Universal Robots URScript: 31-pallet_working.script

def P31pallet_working():
  set_standard_analog_input_domain(0, 1)
  set_standard_analog_input_domain(1, 1)
  set_tool_analog_input_domain(0, 1)
  set_tool_analog_input_domain(1, 1)
  set_analog_outputdomain(0, 0)
  set_analog_outputdomain(1, 0)
  set_tool_voltage(0)
  set_tcp(p[0.0,0.0,0.0,0.0,0.0,0.0])
  set_payload(0.0)
  set_gravity([0.0, 0.0, 9.82])
  global cnt_1=0
  $ 1 "BeforeStart"
  $ 2 "MoveJ"
  $ 3 "home"
  movej([-1.5531271160755855, -1.3695928511239472, -1.6775720824016744, -1.6897506072074169, 1.5962951182804097, 0.016572788116811236], a=1.3962634015954636, v=1.0471975511965976)
  $ 4 "cnt_1≔5"
  global cnt_1=5
  while (True):
    $ 5 "机器人程序"
    $ 6 "托盘"
    cnt_1_x = cnt_1 % 6
    cnt_1_y = floor(cnt_1 / 6)
    u20301u23039_1 = interpolate_pose(interpolate_pose(p[-.099999969066, -.400000054028, .199999960922, -.001221099554, 3.116276478707, .038892320958], p[-.100000003377, -.199999964388, .199999987920, -.001220853457, 3.116276502675, .038892110509], cnt_1_x/5), interpolate_pose(p[.100000089847, -.399999929680, .199999839637, -.001221229174, 3.116276825726, .038892683103], p[.100000030650, -.199999976799, .200000020249, -.001220905867, 3.116276536037, .038892034429],cnt_1_x/5), cnt_1_y/3)
    if (cnt_1 >= 23):
      cnt_1 = 0
    else:
      cnt_1 = cnt_1 + 1
    end
    $ 13 "方式"
    movel(pose_trans(u20301u23039_1, pose_trans(pose_inv(p[-.099999969066, -.400000054028, .199999960922, -.001221099554, 3.116276478707, .038892320958]),p[-.099999970101, -.399999995469, .304818609093, -.001221099554, 3.116276478707, .038892320958])), a=1.2, v=0.25)
    $ 14 "模式点_1"
    movel(u20301u23039_1, a=1.2, v=0.25)
    $ 15 "设置"
    $ 16 "等待: 0"
    $ 17 "退出"
    movel(pose_trans(u20301u23039_1, pose_trans(pose_inv(p[-.099999969066, -.400000054028, .199999960922, -.001221099554, 3.116276478707, .038892320958]),p[-.099999970101, -.399999995469, .304818609093, -.001221099554, 3.116276478707, .038892320958])), a=1.2, v=0.25)
    $ 18 "MoveJ"
    $ 19 "home"
    movej([-1.5531271160755855, -1.3695928511239472, -1.6775720824016744, -1.6897506072074169, 1.5962951182804097, 0.016572788116811236], a=1.3962634015954636, v=1.0471975511965976)
    $ 20 "pick_up"
    movej([0.10491021715125842, -1.4657920746551412, -2.143578449623652, -1.1275450164569616, 1.5962951182776492, 0.01657278801032042], a=1.3962634015954636, v=1.0471975511965976)
    $ 21 "MoveL"
    $ 22 "pick"
    movel([0.10491021708313425, -1.7172361101439613, -2.325250094224021, -0.6944293363695415, 1.5962951182758853, 0.016572787942196247], a=1.2, v=0.25)
    $ 23 "pick_up"
    movel([0.10491021715125842, -1.4657920746551412, -2.143578449623652, -1.1275450164569616, 1.5962951182776492, 0.01657278801032042], a=1.2, v=0.25)
    $ 24 "MoveJ"
    $ 25 "home"
    movej([-1.5531271160755855, -1.3695928511239472, -1.6775720824016744, -1.6897506072074169, 1.5962951182804097, 0.016572788116811236], a=1.3962634015954636, v=1.0471975511965976)
  end
end
